{attribute 'reflection'}
FUNCTION_BLOCK PUBLIC FB_DevHDAnalogInputScaled EXTENDS FB_DevHDAnalogInput
VAR_INPUT
END_VAR
VAR_OUTPUT
END_VAR
VAR
	fGainFactor 	: LREAL	:= 1	;
	nOfset			: DINT	:= 0	;
END_VAR

SUPER^(refFbFault := refFbFault);

METHOD ExecSetFeedback : BOOL
VAR
	nCalibValue	: DINT ; 
END_VAR
// Offset 
IF bCmdSimulate THEN 
	nCalibValue := fSimValue + nOfset ;
ELSE
	nCalibValue := inHwInput + nOfset ;
END_IF

fValue := DINT_TO_LREAL(nCalibValue) / fGainFactor;
END_METHOD

METHOD PUBLIC SetScaling : BOOL 
VAR_INPUT
	fMaxValue	: LREAL ; 	// Maximum input value after scaling, e.g. 100%, 0 = no scaling (gain = hardware limit / fMaxValue)  
	fOfset		: LREAL ;	// offset value (fvalue = (gain * hwvalue) + fOfset)
END_VAR
// calculate gain 
IF fMaxValue =0 THEN 
	fGainFactor := 1 ;
ELSE 
	fGainFactor := nLimitMax / fMaxValue ;
END_IF

nOfset := LREAL_TO_DINT(fOfset * fGainFactor) ;

SetScaling := TRUE ;
END_METHOD

END_FUNCTION_BLOCK

(* stored: Version 1.1.0.1, ProductVersion 3.1.4024.5
   POU FB_DevHDAnalogInputScaled: Id {1d5348c2-1ecf-04c7-34d9-8f2fb7f7f54c}, SpecialFunc None
   Method ExecSetFeedback: Id {ba1246d6-0b89-032f-1cee-0b644ffdc5ff}
   Method SetScaling: Id {0357e09f-11ea-0ea7-2fd6-dab3997dc380} *)
